TYPE TcoSmartFunctionKitStatus_v_4_x_x : STRUCT
    ActionDescription : STRING(100);
    ResponseStatus : TcoSmartFunctionKitResponse_v_4_x_x;
    NotificationId : UINT;
    NotificationToDisplay : eTcoSmartFunctionKitStatusInformation_v_4_x_x;
    NotificationPosition : REAL;
    NotificationVelocity : REAL;
    NotificationForce : REAL;
    DigitalIoMapping : DWORD;
    VirtualIo : DWORD;
END_STRUCT
END_TYPE

(* stored: Version 1.1.0.1, ProductVersion 3.1.4024.11
   DUT TcoSmartFunctionKitStatus_v_4_x_x: Id {b670224a-a0c6-4af9-849f-e8cab4f5328e} *)
